TYPE ENUM_CarrierPos :
(
	Left 	:= 1,
	Right 	:= 2
)UINT;
END_TYPE

(* stored: Version 1.1.0.1, ProductVersion 3.1.4024.12
   DUT ENUM_CarrierPos: Id {a55ef211-4820-49b5-99d1-239944ccc67c} *)
